// TwinCAT 3 PLC project IO
// ProgramVersion: 3.1.4024.0
// libraries:
//   Tc2_Standard, * (Beckhoff Automation GmbH)
//   Tc2_System, * (Beckhoff Automation GmbH)
//   Tc3_Module, * (Beckhoff Automation GmbH)
//   TcUnit, * (www.tcunit.org)
// project tree:
//   TESTS/ PRG_TESTS.TcPOU
//   TESTS/Test suites/ FB_SUT_Tests.TcPOU (not stored)
// real-time tasks:
//   TASK TestsTask: cycle T#10ms, priority 20, ADS port 350

// ---- TESTS/PRG_TESTS.TcPOU
PROGRAM PRG_TESTS

(* Instantiate test suites here. Naming convention for tests should be a suffix with _Tests.
Good practice for creating test methods is to end them with _test as well. *)
VAR
	fbSUT_Tests	: FB_SUT_Tests;
END_VAR

// Run tests in paralel
TcUnit.RUN();

// Run tests in sequence, one after the other. Uncomment if required.
// TcUnit.RUN_IN_SEQUENCE();

END_PROGRAM
